(* Logix 5000 project; controller cal1615 1756-L62 rev 20.11; software revision 20.05; part 66 of 82 *)
(* tags used below, declared in another part *)
   FAULT : BOOL;   // Fault AFI
   HMI : BOOL;   // AFI HMI
   p01r09_pb_global_reset : BOOL;   // System Modes PB: Global Fault Reset
   p27_ao_dia_a : REAL;   // Lower Poly Letoff Analog Input Letoff A Diameter
   p27_ao_dia_b : REAL;   // Lower Poly Letoff Analog Input Letoff B Diameter
   p27_dint_to_hmi : DINT[16];   // Lower Poly Letoff Alarms
   p27_real_to_hmi : REAL[112];   // Winder Real to HMI
   p27r01 : routine;   // Winder Main
   p27r06 : routine;   // Winder Real to HMI
   p27r06_timer_fault : TIMER[4];   // Winder Real to HMI Fault Delay
   p27r06_timer_warning : TIMER[4];   // Winder Real to HMI Warning Delay
   p27r07 : routine;   // Winder Alarms
   p27r07_timer_fault : TIMER[4];   // Winder Alarms Fault Delay
   p27r07_timer_warning : TIMER[4];   // Winder Alarms Warning Delay
   p27r08 : routine;   // Winder Warnings
   p27r08_timer_fault : TIMER[4];   // Winder Warnings Fault Delay
   p27r08_timer_warning : TIMER[4];   // Winder Warnings Warning Delay
(* P27_Lower_Poly_Letoff, continued *)

ROUTINE R06_Real_to_HMI   (* ladder *)
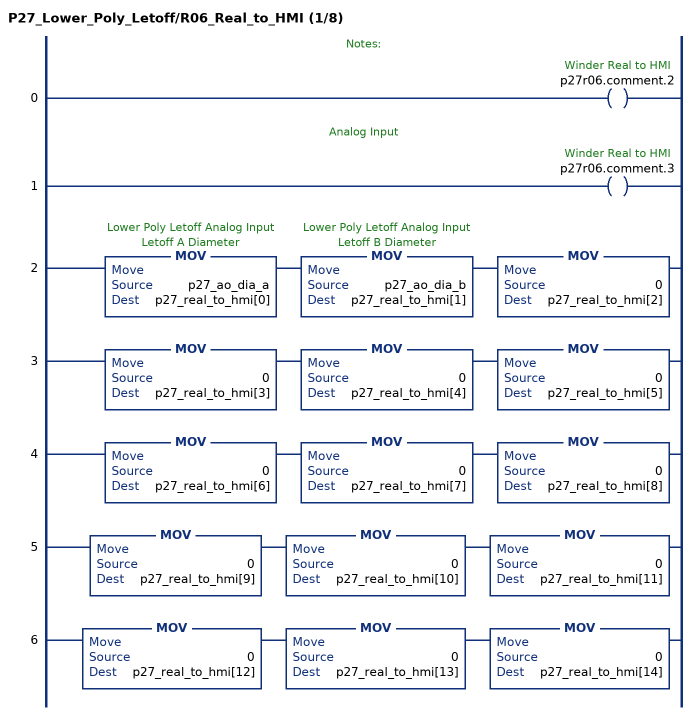
   // Notes:
   0: OTE(p27r06.comment.2);
   // Analog Input
   1: OTE(p27r06.comment.3);
   2: MOV(p27_ao_dia_a,p27_real_to_hmi[0])MOV(p27_ao_dia_b,p27_real_to_hmi[1])MOV(0,p27_real_to_hmi[2]);
   3: MOV(0,p27_real_to_hmi[3])MOV(0,p27_real_to_hmi[4])MOV(0,p27_real_to_hmi[5]);
   4: MOV(0,p27_real_to_hmi[6])MOV(0,p27_real_to_hmi[7])MOV(0,p27_real_to_hmi[8]);
   5: MOV(0,p27_real_to_hmi[9])MOV(0,p27_real_to_hmi[10])MOV(0,p27_real_to_hmi[11]);
   6: MOV(0,p27_real_to_hmi[12])MOV(0,p27_real_to_hmi[13])MOV(0,p27_real_to_hmi[14]);
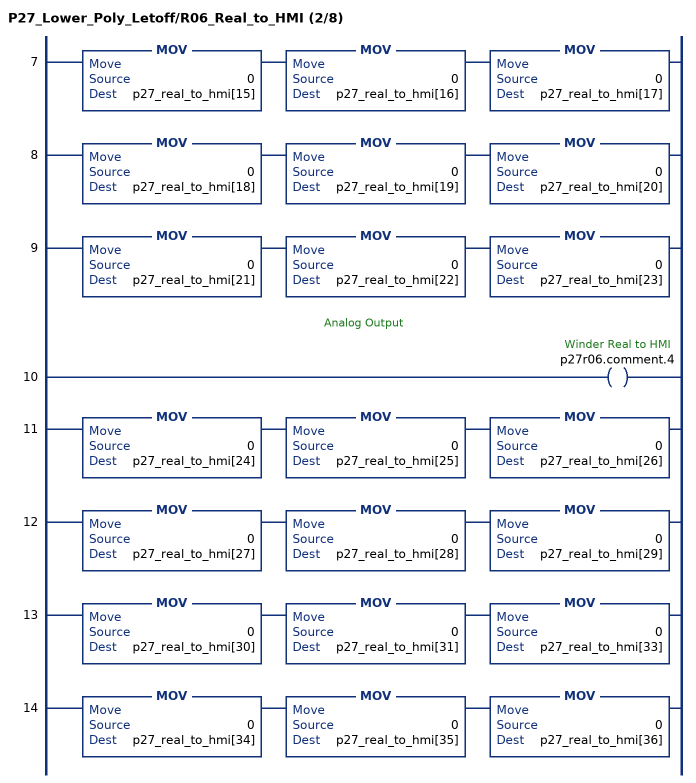
   7: MOV(0,p27_real_to_hmi[15])MOV(0,p27_real_to_hmi[16])MOV(0,p27_real_to_hmi[17]);
   8: MOV(0,p27_real_to_hmi[18])MOV(0,p27_real_to_hmi[19])MOV(0,p27_real_to_hmi[20]);
   9: MOV(0,p27_real_to_hmi[21])MOV(0,p27_real_to_hmi[22])MOV(0,p27_real_to_hmi[23]);
   // Analog Output
   10: OTE(p27r06.comment.4);
   11: MOV(0,p27_real_to_hmi[24])MOV(0,p27_real_to_hmi[25])MOV(0,p27_real_to_hmi[26]);
   12: MOV(0,p27_real_to_hmi[27])MOV(0,p27_real_to_hmi[28])MOV(0,p27_real_to_hmi[29]);
   13: MOV(0,p27_real_to_hmi[30])MOV(0,p27_real_to_hmi[31])MOV(0,p27_real_to_hmi[33]);
   14: MOV(0,p27_real_to_hmi[34])MOV(0,p27_real_to_hmi[35])MOV(0,p27_real_to_hmi[36]);
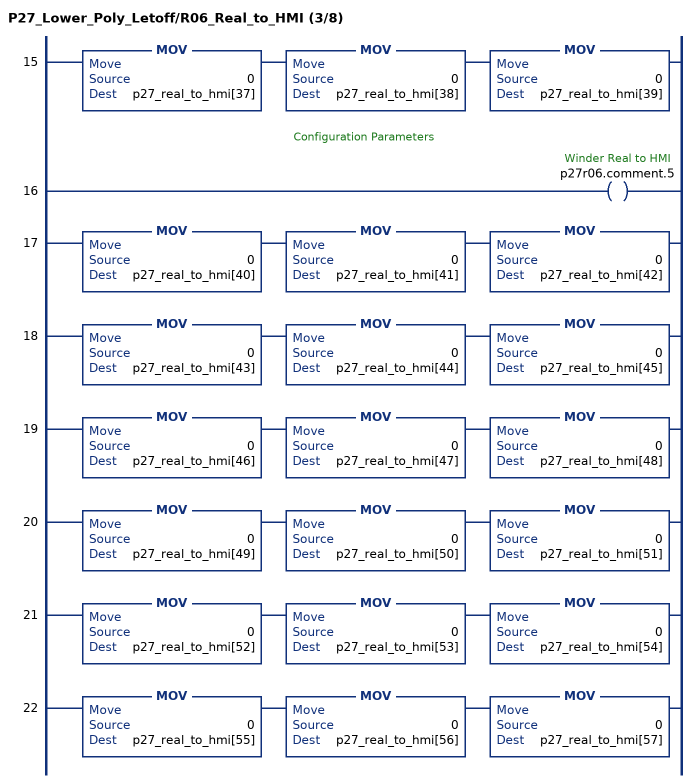
   15: MOV(0,p27_real_to_hmi[37])MOV(0,p27_real_to_hmi[38])MOV(0,p27_real_to_hmi[39]);
   // Configuration Parameters
   16: OTE(p27r06.comment.5);
   17: MOV(0,p27_real_to_hmi[40])MOV(0,p27_real_to_hmi[41])MOV(0,p27_real_to_hmi[42]);
   18: MOV(0,p27_real_to_hmi[43])MOV(0,p27_real_to_hmi[44])MOV(0,p27_real_to_hmi[45]);
   19: MOV(0,p27_real_to_hmi[46])MOV(0,p27_real_to_hmi[47])MOV(0,p27_real_to_hmi[48]);
   20: MOV(0,p27_real_to_hmi[49])MOV(0,p27_real_to_hmi[50])MOV(0,p27_real_to_hmi[51]);
   21: MOV(0,p27_real_to_hmi[52])MOV(0,p27_real_to_hmi[53])MOV(0,p27_real_to_hmi[54]);
   22: MOV(0,p27_real_to_hmi[55])MOV(0,p27_real_to_hmi[56])MOV(0,p27_real_to_hmi[57]);
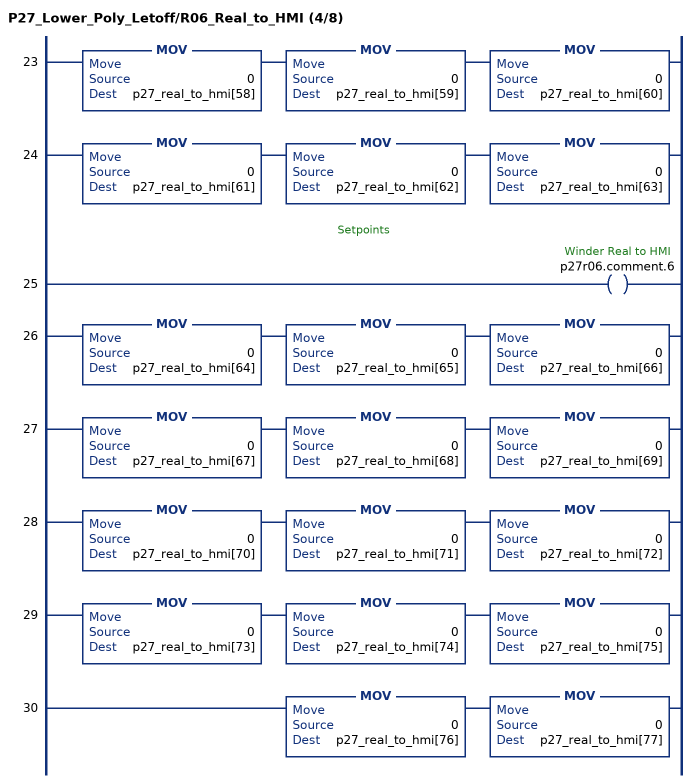
   23: MOV(0,p27_real_to_hmi[58])MOV(0,p27_real_to_hmi[59])MOV(0,p27_real_to_hmi[60]);
   24: MOV(0,p27_real_to_hmi[61])MOV(0,p27_real_to_hmi[62])MOV(0,p27_real_to_hmi[63]);
   // Setpoints
   25: OTE(p27r06.comment.6);
   26: MOV(0,p27_real_to_hmi[64])MOV(0,p27_real_to_hmi[65])MOV(0,p27_real_to_hmi[66]);
   27: MOV(0,p27_real_to_hmi[67])MOV(0,p27_real_to_hmi[68])MOV(0,p27_real_to_hmi[69]);
   28: MOV(0,p27_real_to_hmi[70])MOV(0,p27_real_to_hmi[71])MOV(0,p27_real_to_hmi[72]);
   29: MOV(0,p27_real_to_hmi[73])MOV(0,p27_real_to_hmi[74])MOV(0,p27_real_to_hmi[75]);
   30: MOV(0,p27_real_to_hmi[76])MOV(0,p27_real_to_hmi[77]);
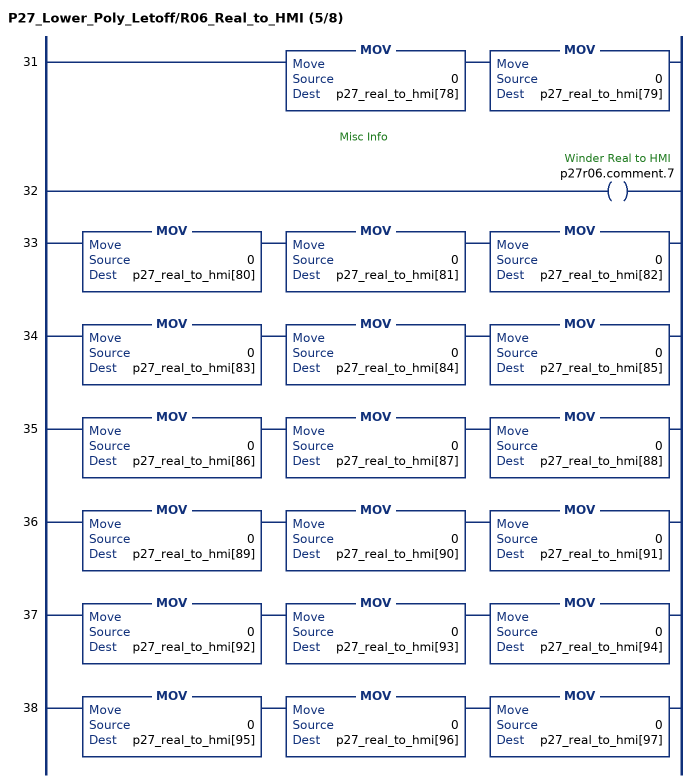
   31: MOV(0,p27_real_to_hmi[78])MOV(0,p27_real_to_hmi[79]);
   // Misc Info
   32: OTE(p27r06.comment.7);
   33: MOV(0,p27_real_to_hmi[80])MOV(0,p27_real_to_hmi[81])MOV(0,p27_real_to_hmi[82]);
   34: MOV(0,p27_real_to_hmi[83])MOV(0,p27_real_to_hmi[84])MOV(0,p27_real_to_hmi[85]);
   35: MOV(0,p27_real_to_hmi[86])MOV(0,p27_real_to_hmi[87])MOV(0,p27_real_to_hmi[88]);
   36: MOV(0,p27_real_to_hmi[89])MOV(0,p27_real_to_hmi[90])MOV(0,p27_real_to_hmi[91]);
   37: MOV(0,p27_real_to_hmi[92])MOV(0,p27_real_to_hmi[93])MOV(0,p27_real_to_hmi[94]);
   38: MOV(0,p27_real_to_hmi[95])MOV(0,p27_real_to_hmi[96])MOV(0,p27_real_to_hmi[97]);
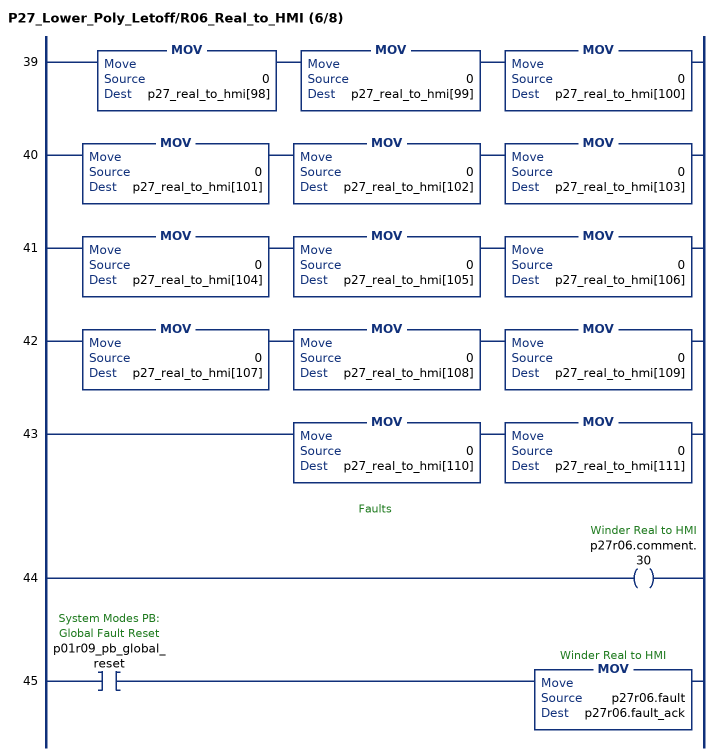
   39: MOV(0,p27_real_to_hmi[98])MOV(0,p27_real_to_hmi[99])MOV(0,p27_real_to_hmi[100]);
   40: MOV(0,p27_real_to_hmi[101])MOV(0,p27_real_to_hmi[102])MOV(0,p27_real_to_hmi[103]);
   41: MOV(0,p27_real_to_hmi[104])MOV(0,p27_real_to_hmi[105])MOV(0,p27_real_to_hmi[106]);
   42: MOV(0,p27_real_to_hmi[107])MOV(0,p27_real_to_hmi[108])MOV(0,p27_real_to_hmi[109]);
   43: MOV(0,p27_real_to_hmi[110])MOV(0,p27_real_to_hmi[111]);
   // Faults
   44: OTE(p27r06.comment.30);
   45: XIC(p01r09_pb_global_reset)MOV(p27r06.fault,p27r06.fault_ack);
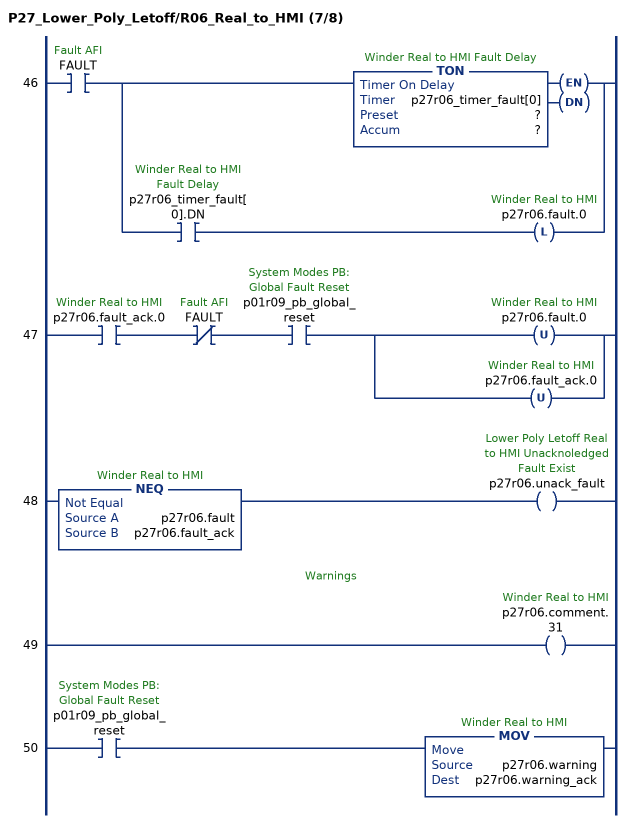
   46: XIC(FAULT)[TON(p27r06_timer_fault[0],?,?) ,XIC(p27r06_timer_fault[0].DN) OTL(p27r06.fault.0) ];
   47: XIC(p27r06.fault_ack.0)XIO(FAULT)XIC(p01r09_pb_global_reset)[OTU(p27r06.fault.0) ,OTU(p27r06.fault_ack.0) ];
   48: NEQ(p27r06.fault,p27r06.fault_ack)OTE(p27r06.unack_fault);
   // Warnings
   49: OTE(p27r06.comment.31);
   50: XIC(p01r09_pb_global_reset)MOV(p27r06.warning,p27r06.warning_ack);
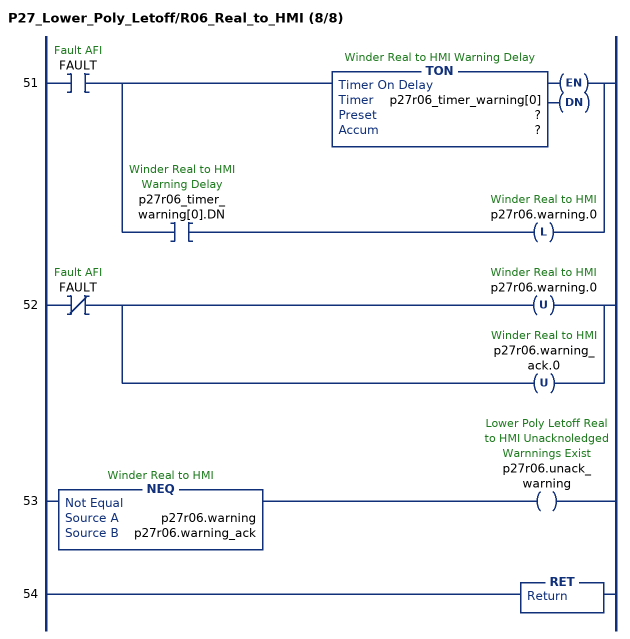
   51: XIC(FAULT)[TON(p27r06_timer_warning[0],?,?) ,XIC(p27r06_timer_warning[0].DN) OTL(p27r06.warning.0) ];
   52: XIO(FAULT)[OTU(p27r06.warning.0) ,OTU(p27r06.warning_ack.0) ];
   53: NEQ(p27r06.warning,p27r06.warning_ack)OTE(p27r06.unack_warning);
   54: RET();
END_ROUTINE

ROUTINE R07_Alarms   (* ladder *)
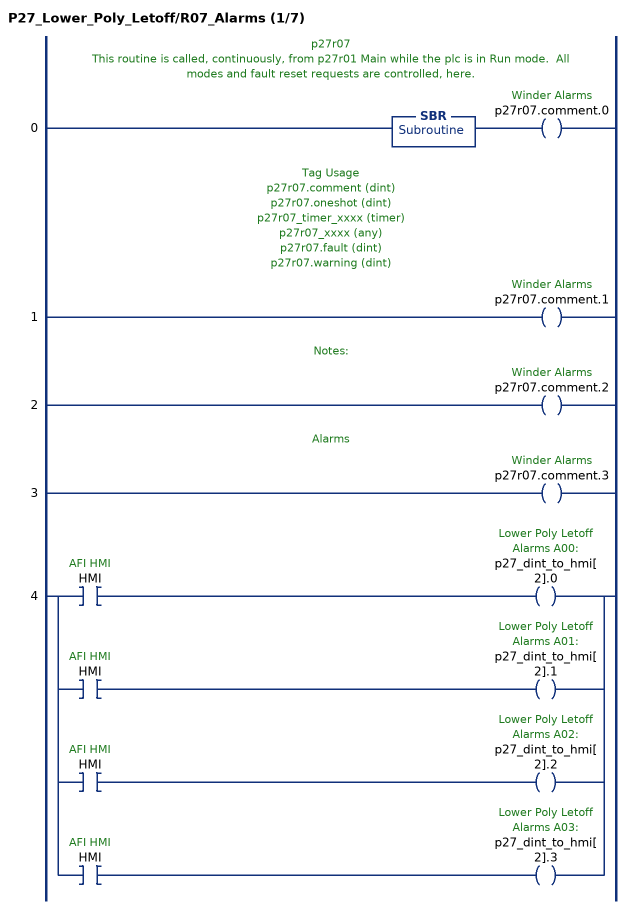
   // p27r07
   // This routine is called, continuously, from p27r01 Main while the plc is in Run mode.  All modes and fault reset requests are controlled, here.
   0: SBR()OTE(p27r07.comment.0);
   // Tag Usage
   // p27r07.comment (dint)
   // p27r07.oneshot (dint)
   // p27r07_timer_xxxx (timer)
   // p27r07_xxxx (any)
   // p27r07.fault (dint)
   // p27r07.warning (dint)
   1: OTE(p27r07.comment.1);
   // Notes:
   2: OTE(p27r07.comment.2);
   // Alarms
   3: OTE(p27r07.comment.3);
   4: [XIC(HMI) OTE(p27_dint_to_hmi[2].0) ,XIC(HMI) OTE(p27_dint_to_hmi[2].1) ,XIC(HMI) OTE(p27_dint_to_hmi[2].2) ,XIC(HMI) OTE(p27_dint_to_hmi[2].3) ];
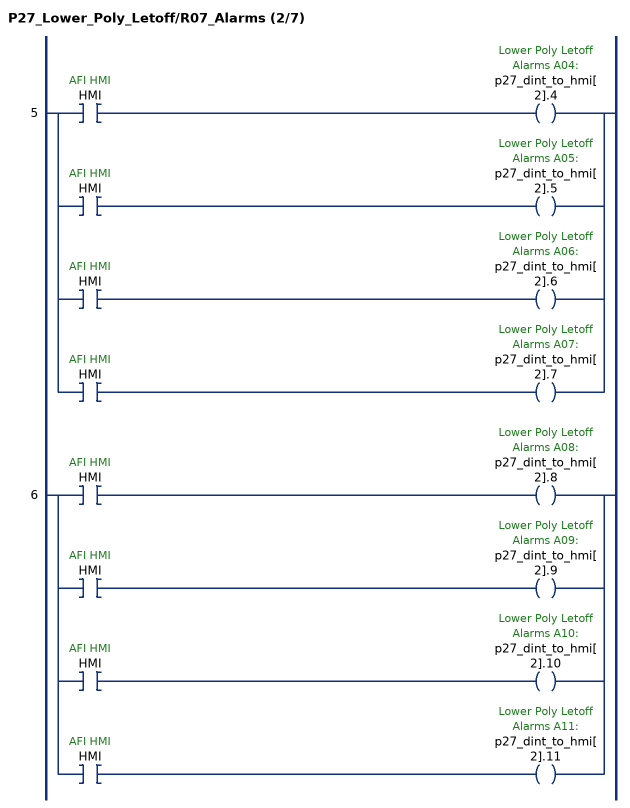
   5: [XIC(HMI) OTE(p27_dint_to_hmi[2].4) ,XIC(HMI) OTE(p27_dint_to_hmi[2].5) ,XIC(HMI) OTE(p27_dint_to_hmi[2].6) ,XIC(HMI) OTE(p27_dint_to_hmi[2].7) ];
   6: [XIC(HMI) OTE(p27_dint_to_hmi[2].8) ,XIC(HMI) OTE(p27_dint_to_hmi[2].9) ,XIC(HMI) OTE(p27_dint_to_hmi[2].10) ,XIC(HMI) OTE(p27_dint_to_hmi[2].11) ];
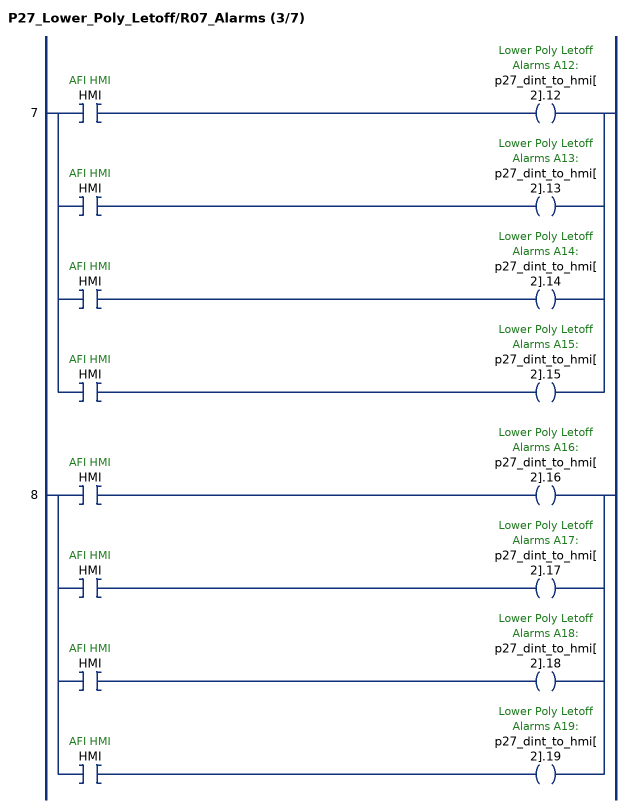
   7: [XIC(HMI) OTE(p27_dint_to_hmi[2].12) ,XIC(HMI) OTE(p27_dint_to_hmi[2].13) ,XIC(HMI) OTE(p27_dint_to_hmi[2].14) ,XIC(HMI) OTE(p27_dint_to_hmi[2].15) ];
   8: [XIC(HMI) OTE(p27_dint_to_hmi[2].16) ,XIC(HMI) OTE(p27_dint_to_hmi[2].17) ,XIC(HMI) OTE(p27_dint_to_hmi[2].18) ,XIC(HMI) OTE(p27_dint_to_hmi[2].19) ];
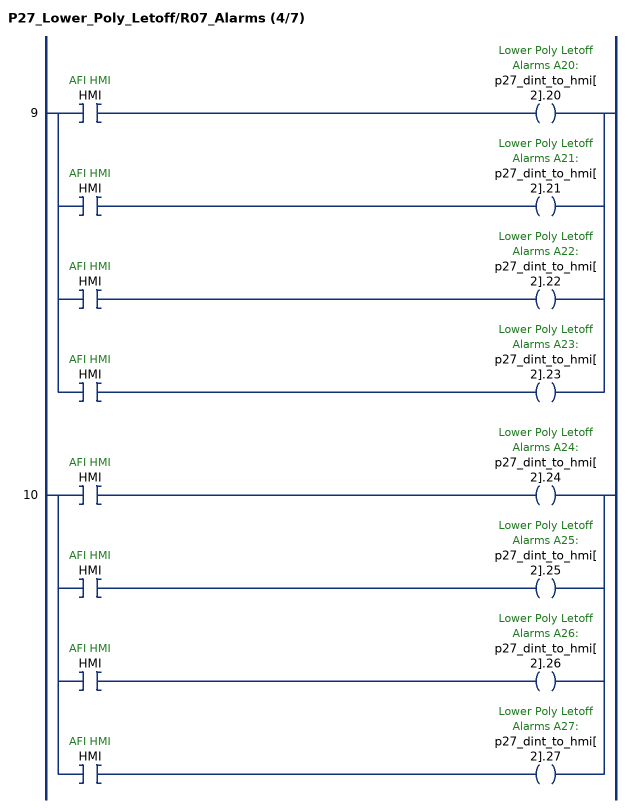
   9: [XIC(HMI) OTE(p27_dint_to_hmi[2].20) ,XIC(HMI) OTE(p27_dint_to_hmi[2].21) ,XIC(HMI) OTE(p27_dint_to_hmi[2].22) ,XIC(HMI) OTE(p27_dint_to_hmi[2].23) ];
   10: [XIC(HMI) OTE(p27_dint_to_hmi[2].24) ,XIC(HMI) OTE(p27_dint_to_hmi[2].25) ,XIC(HMI) OTE(p27_dint_to_hmi[2].26) ,XIC(HMI) OTE(p27_dint_to_hmi[2].27) ];
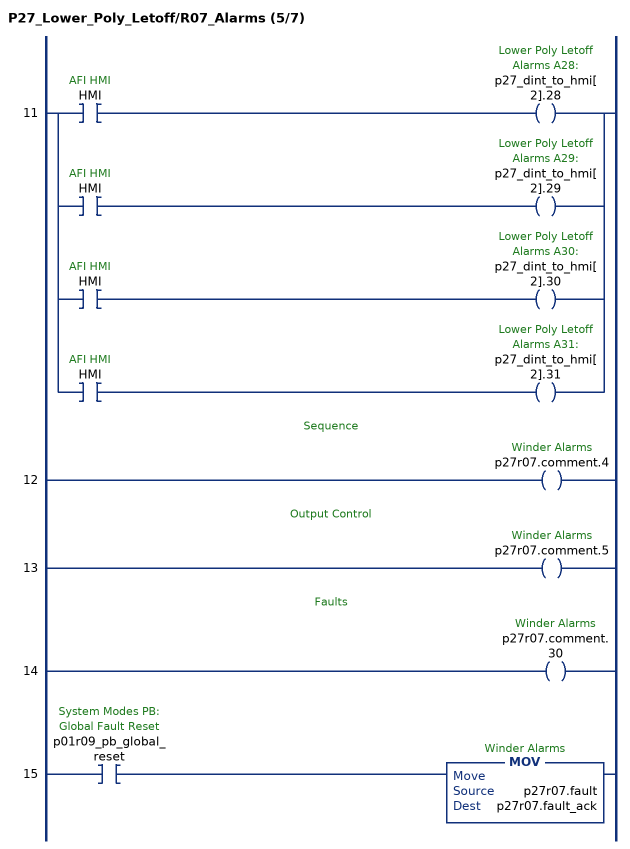
   11: [XIC(HMI) OTE(p27_dint_to_hmi[2].28) ,XIC(HMI) OTE(p27_dint_to_hmi[2].29) ,XIC(HMI) OTE(p27_dint_to_hmi[2].30) ,XIC(HMI) OTE(p27_dint_to_hmi[2].31) ];
   // Sequence
   12: OTE(p27r07.comment.4);
   // Output Control
   13: OTE(p27r07.comment.5);
   // Faults
   14: OTE(p27r07.comment.30);
   15: XIC(p01r09_pb_global_reset)MOV(p27r07.fault,p27r07.fault_ack);
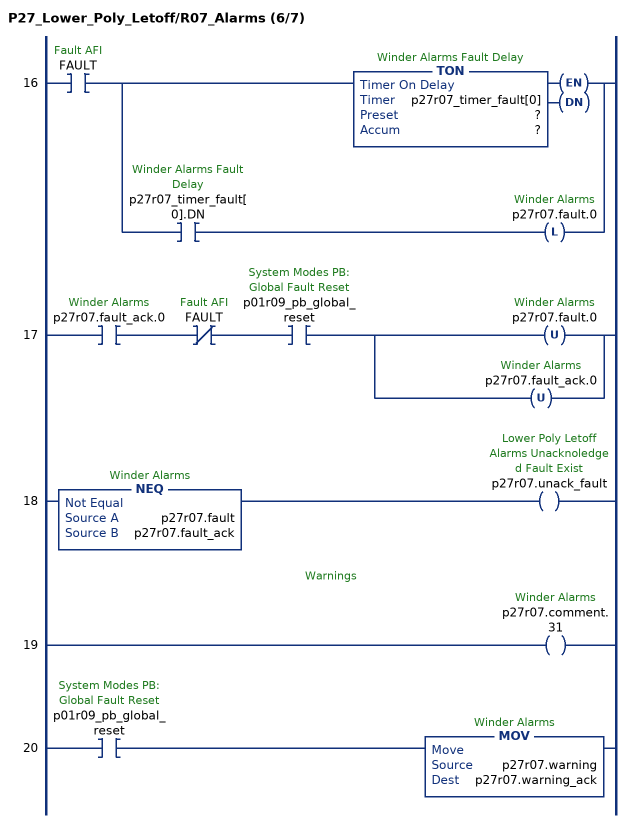
   16: XIC(FAULT)[TON(p27r07_timer_fault[0],?,?) ,XIC(p27r07_timer_fault[0].DN) OTL(p27r07.fault.0) ];
   17: XIC(p27r07.fault_ack.0)XIO(FAULT)XIC(p01r09_pb_global_reset)[OTU(p27r07.fault.0) ,OTU(p27r07.fault_ack.0) ];
   18: NEQ(p27r07.fault,p27r07.fault_ack)OTE(p27r07.unack_fault);
   // Warnings
   19: OTE(p27r07.comment.31);
   20: XIC(p01r09_pb_global_reset)MOV(p27r07.warning,p27r07.warning_ack);
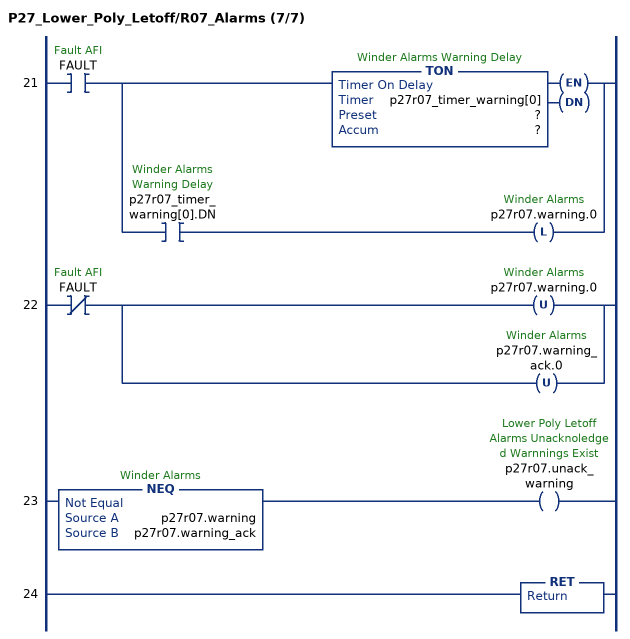
   21: XIC(FAULT)[TON(p27r07_timer_warning[0],?,?) ,XIC(p27r07_timer_warning[0].DN) OTL(p27r07.warning.0) ];
   22: XIO(FAULT)[OTU(p27r07.warning.0) ,OTU(p27r07.warning_ack.0) ];
   23: NEQ(p27r07.warning,p27r07.warning_ack)OTE(p27r07.unack_warning);
   24: RET();
END_ROUTINE

ROUTINE R08_Warnings   (* ladder *)
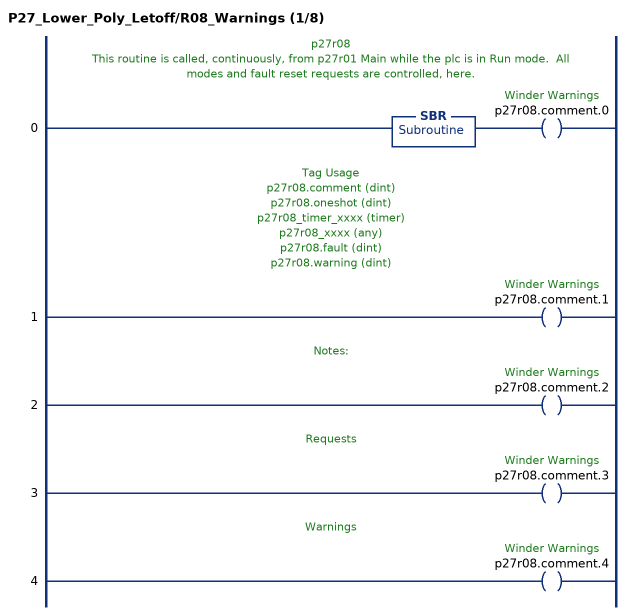
   // p27r08
   // This routine is called, continuously, from p27r01 Main while the plc is in Run mode.  All modes and fault reset requests are controlled, here.
   0: SBR()OTE(p27r08.comment.0);
   // Tag Usage
   // p27r08.comment (dint)
   // p27r08.oneshot (dint)
   // p27r08_timer_xxxx (timer)
   // p27r08_xxxx (any)
   // p27r08.fault (dint)
   // p27r08.warning (dint)
   1: OTE(p27r08.comment.1);
   // Notes:
   2: OTE(p27r08.comment.2);
   // Requests
   3: OTE(p27r08.comment.3);
   // Warnings
   4: OTE(p27r08.comment.4);
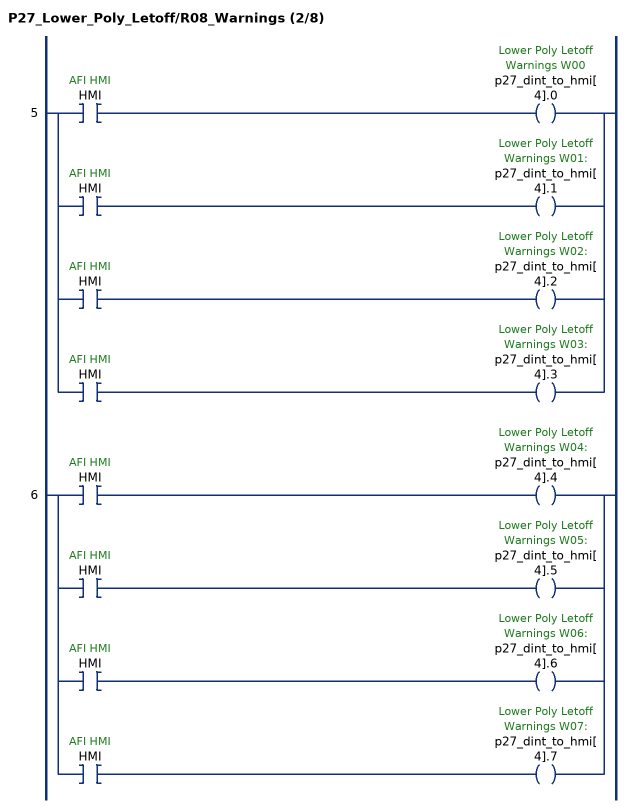
   5: [XIC(HMI) OTE(p27_dint_to_hmi[4].0) ,XIC(HMI) OTE(p27_dint_to_hmi[4].1) ,XIC(HMI) OTE(p27_dint_to_hmi[4].2) ,XIC(HMI) OTE(p27_dint_to_hmi[4].3) ];
   6: [XIC(HMI) OTE(p27_dint_to_hmi[4].4) ,XIC(HMI) OTE(p27_dint_to_hmi[4].5) ,XIC(HMI) OTE(p27_dint_to_hmi[4].6) ,XIC(HMI) OTE(p27_dint_to_hmi[4].7) ];
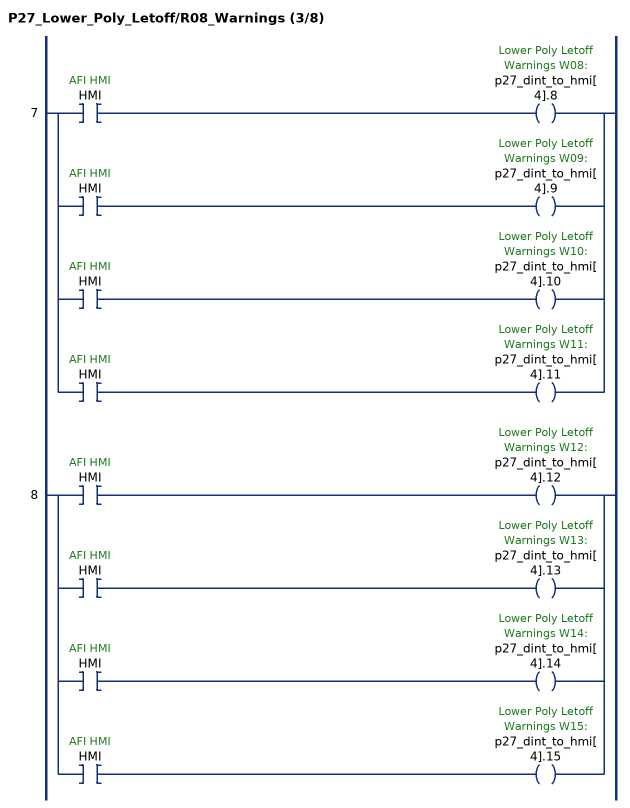
   7: [XIC(HMI) OTE(p27_dint_to_hmi[4].8) ,XIC(HMI) OTE(p27_dint_to_hmi[4].9) ,XIC(HMI) OTE(p27_dint_to_hmi[4].10) ,XIC(HMI) OTE(p27_dint_to_hmi[4].11) ];
   8: [XIC(HMI) OTE(p27_dint_to_hmi[4].12) ,XIC(HMI) OTE(p27_dint_to_hmi[4].13) ,XIC(HMI) OTE(p27_dint_to_hmi[4].14) ,XIC(HMI) OTE(p27_dint_to_hmi[4].15) ];
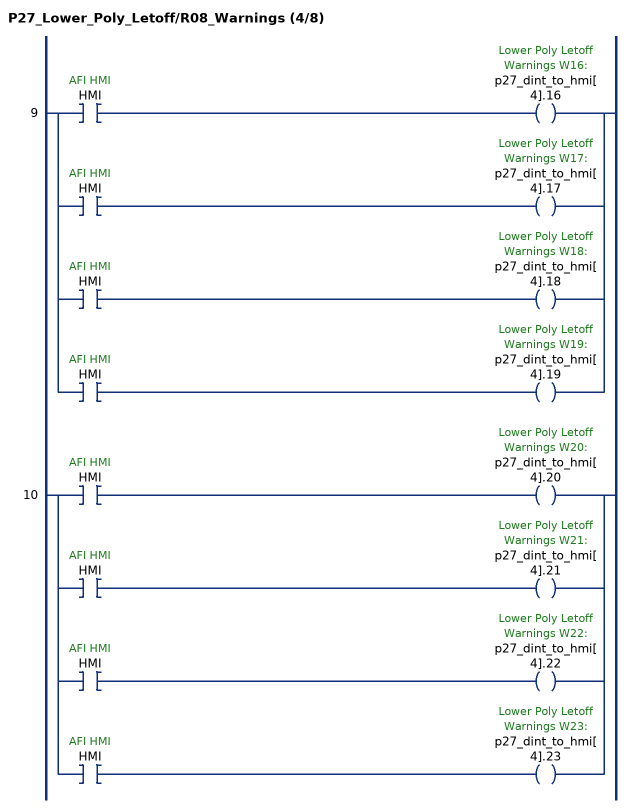
   9: [XIC(HMI) OTE(p27_dint_to_hmi[4].16) ,XIC(HMI) OTE(p27_dint_to_hmi[4].17) ,XIC(HMI) OTE(p27_dint_to_hmi[4].18) ,XIC(HMI) OTE(p27_dint_to_hmi[4].19) ];
   10: [XIC(HMI) OTE(p27_dint_to_hmi[4].20) ,XIC(HMI) OTE(p27_dint_to_hmi[4].21) ,XIC(HMI) OTE(p27_dint_to_hmi[4].22) ,XIC(HMI) OTE(p27_dint_to_hmi[4].23) ];
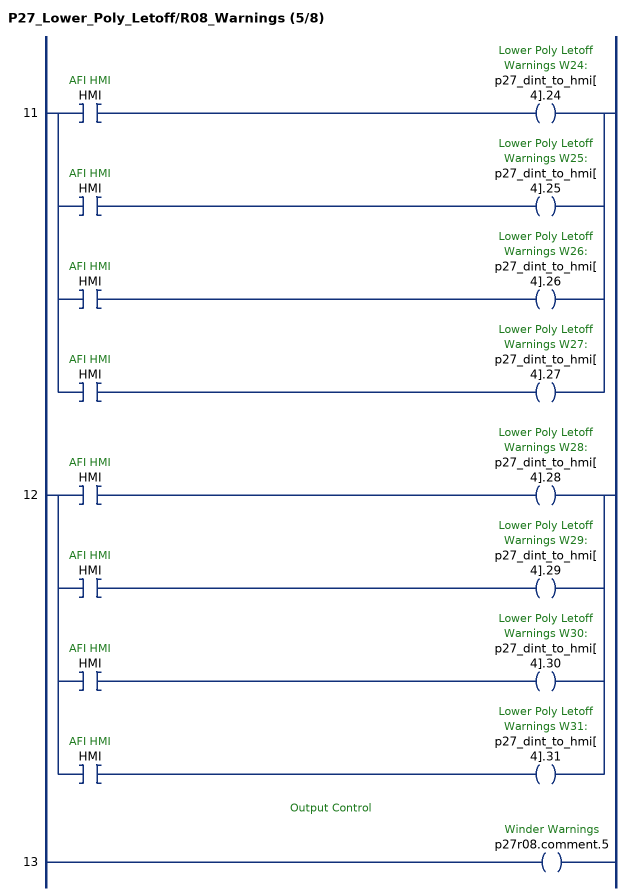
   11: [XIC(HMI) OTE(p27_dint_to_hmi[4].24) ,XIC(HMI) OTE(p27_dint_to_hmi[4].25) ,XIC(HMI) OTE(p27_dint_to_hmi[4].26) ,XIC(HMI) OTE(p27_dint_to_hmi[4].27) ];
   12: [XIC(HMI) OTE(p27_dint_to_hmi[4].28) ,XIC(HMI) OTE(p27_dint_to_hmi[4].29) ,XIC(HMI) OTE(p27_dint_to_hmi[4].30) ,XIC(HMI) OTE(p27_dint_to_hmi[4].31) ];
   // Output Control
   13: OTE(p27r08.comment.5);
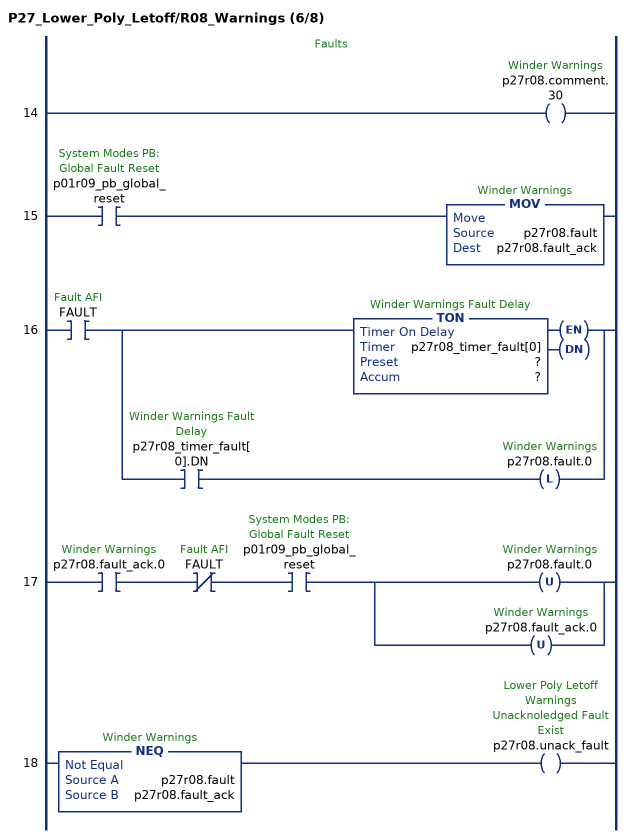
   // Faults
   14: OTE(p27r08.comment.30);
   15: XIC(p01r09_pb_global_reset)MOV(p27r08.fault,p27r08.fault_ack);
   16: XIC(FAULT)[TON(p27r08_timer_fault[0],?,?) ,XIC(p27r08_timer_fault[0].DN) OTL(p27r08.fault.0) ];
   17: XIC(p27r08.fault_ack.0)XIO(FAULT)XIC(p01r09_pb_global_reset)[OTU(p27r08.fault.0) ,OTU(p27r08.fault_ack.0) ];
   18: NEQ(p27r08.fault,p27r08.fault_ack)OTE(p27r08.unack_fault);
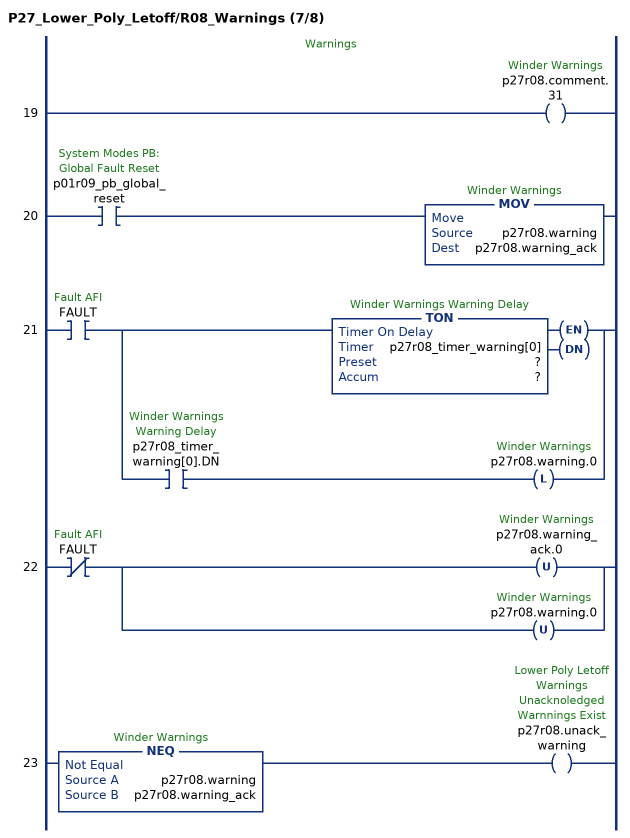
   // Warnings
   19: OTE(p27r08.comment.31);
   20: XIC(p01r09_pb_global_reset)MOV(p27r08.warning,p27r08.warning_ack);
   21: XIC(FAULT)[TON(p27r08_timer_warning[0],?,?) ,XIC(p27r08_timer_warning[0].DN) OTL(p27r08.warning.0) ];
   22: XIO(FAULT)[OTU(p27r08.warning_ack.0) ,OTU(p27r08.warning.0) ];
   23: NEQ(p27r08.warning,p27r08.warning_ack)OTE(p27r08.unack_warning);
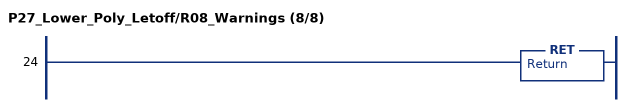
   24: RET();
END_ROUTINE
